// This function has been automatically generated from the project information.
{attribute 'signature_flag' := '1073741824'}
{attribute 'TcGenerated'}
{attribute 'no-analysis'}
FUNCTION F_GetTitle : WSTRING
VAR_INPUT
	
END_VAR

F_GetTitle := "CNM_CycleManager";

END_FUNCTION

(* stored: Version 1.1.0.1
   POU F_GetTitle: Id {78a2157f-74e0-42f7-bda3-b12a6921be96}, SpecialFunc None *)
